TYPE Cnv_Level_Inputs_DUT :
STRUCT
	Cnv1_Inputs:	Buffer_Cnv_Inputs_DUT;
	Cnv2_Inputs:	Buffer_Cnv_Inputs_DUT;
END_STRUCT
END_TYPE

(* stored: Version 1.1.0.1
   DUT Cnv_Level_Inputs_DUT: Id {5f4568dd-6447-4d4d-85e1-3bf13cad1094} *)
